TEXTLIST LineLoadClose
  0 = '主流线&缓存线上料' | Chinese: '主流线&缓存线上料' | English: 'LineLoad_None' | Vietnamese: 'LineLoad_None'
  1 = '主流线上料关闭' | Chinese: '主流线上料关闭' | English: 'Line0Close' | Vietnamese: 'Line1Close'
  2 = '缓存线上料关闭' | Chinese: '缓存线上料关闭' | English: 'LineAcquireClose' | Vietnamese: 'LineAcquireClose'
   = ''
END_TEXTLIST

(* stored: Version 1.1.0.1, ProductVersion 3.1.4024.3
   TextList LineLoadClose: Id {d63b00bf-042e-4bad-b7d3-7741a0326ed6} *)
